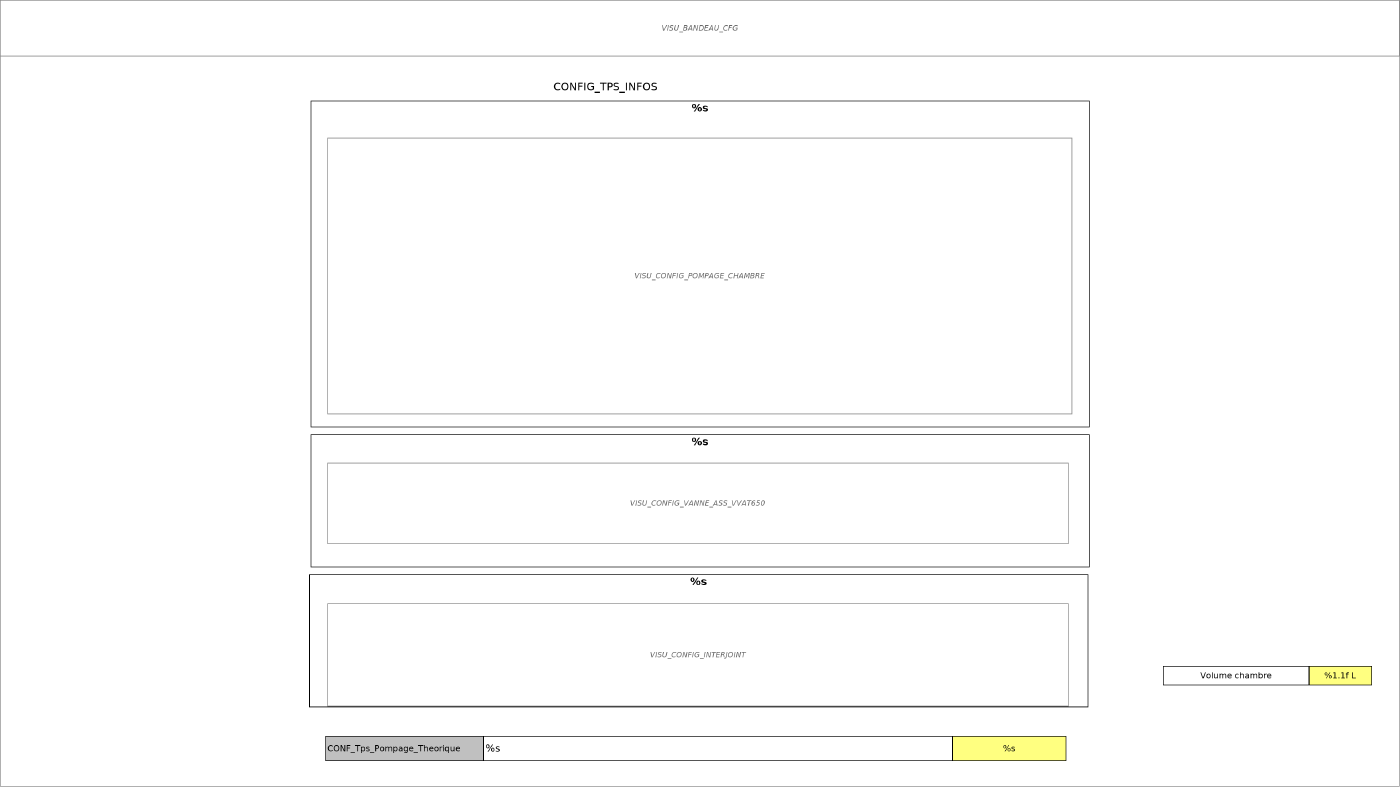
VISUALIZATION VISU_CONFIG_POMPAGE  // 1920x1080, background image fond_blanc_1280_1024
    RoundedRectangle (426,138 1068x448), "%s", text list: 'TextList_Config_Pompage', text index: 0
    Frame (0,0 1920x77)
        shows VISU_BANDEAU_CFG()
    Rectangle (756,109 300x20), "CONFIG_TPS_INFOS"
    Rectangle (1595,914 200x26), "Volume chambre"
    Rectangle (1795,914 86x26), "%1.1f L", text variable: Global_Variables.PRG_POMPAGE.POMPAGE.CONF_Volume_Enceinte, input disabled if: NOT Global_Variables.PRG_USER.ACTU_USER.CONF_MACHINE
        OnMouseDown: write the text variable via InputWithLimits
    Frame (449,189 1021x379)
        shows VISU_CONFIG_POMPAGE_CHAMBRE(m_Input_PRG_POMPAGE := PRG_POMPAGE)
    RoundedRectangle (426,596 1068x182), "%s", text list: 'TextList_Config_Pompage', text index: 15
    Rectangle (446,1010 217x34), "CONF_Tps_Pompage_Theorique"
    Rectangle (663,1010 643x34), "%s", text list: 'TextList_Config_Pompage', text index: 16
    Rectangle (1306,1010 156x34), "%s", text variable: PRG_POMPAGE.CONF_Tps_Pompage_Theorique, input disabled if: NOT Global_Variables.PRG_USER.ACTU_USER.CONF_MACHINE
        OnMouseDown: write the text variable via InputWithLimits
    RoundedRectangle (424,788 1068x182), "%s", text list: 'TextList_Config_Pompage', text index: 20
    Frame (449,828 1016x141)
        shows VISU_CONFIG_INTERJOINT(m_Input_Pompage := PRG_POMPAGE.POMPAGE)
    Frame (449,635 1016x111)
        shows VISU_CONFIG_VANNE_ASS_VVAT650(m_Input_Vanne := PRG_POMPAGE.POMPAGE.VS11)
END_VISUALIZATION

(* stored: Version 1.1.0.1, ProductVersion 3.1.4026.18
   Visu VISU_CONFIG_POMPAGE: Id {3fd16dc3-5358-42de-89e3-0b81df4ca3c9} *)
